FUNCTION_BLOCK XtsStations
VAR
END_VAR

METHOD InitialiseStation : BOOL
VAR_INPUT
END_VAR
END_METHOD

METHOD StationMover : BOOL
VAR_INPUT
	MoverNumber : INT;
END_VAR
END_METHOD

END_FUNCTION_BLOCK

(* stored: Version 1.1.0.1, ProductVersion 3.1.4024.12
   POU XtsStations: Id {d5315d8a-1ca1-418d-8e57-21a3ecd9efda}, SpecialFunc None
   Method InitialiseStation: Id {3870bfcd-ebc8-4ecd-94a4-5d0ed719be4f}
   Method StationMover: Id {a72c11b4-4d04-46e2-b90d-6d348aace3f3} *)
